Omron Sysmac Studio project asansörsonnnnnnnnnn (Sysmac Studio 1.43.0.9, StandardProject)

# Controller new_Controller_0: NJ501-1500 version 1.42
Units and slaves: Power Supply : NJ-Px3001; CPU : NJ501-1500
Task PrimaryTask (priority 4, period or condition 1000): Program0

PROGRAM Program0
VAR
    buton1 : BOOL;  (* buton1 *)
    buton2 : BOOL;  (* buton2 *)
    butonn : INT;
    buton3 : BOOL;
    kat1 : BOOL;
    sensor : INT;
    kat2 : BOOL;
    kat3 : BOOL;
    motor : INT;
    ileri : BOOL;
    geri : BOOL;
    dizi : ARRAY[0..2] OF INT;
    görev : INT;
    kapiac : BOOL;  (* kapiac *)
    kapikapa : BOOL;  (* kapikapamotor *)
    kapiacilmasüresi : TON;
    a : TIME;
    kapikapanmasüresi : TON;
    b : TIME;
    kapikapalisensör : BOOL;  (* kapikapalisensör *)
    kapiaciksensör : BOOL;  (* kapiaciksensör *)
    kapiacilmasüresi2 : TON;
    c : TIME;
    kapikapanmasüresi2 : TON;
    kapiacilmasüresi1 : TON;
    kapiacilmasüresi3 : TON;
    kapiac2 : BOOL;  (* kapiac2 *)
    kapikapa2 : BOOL;  (* kapikapa2 *)
    kapiac3 : BOOL;  (* kapiac3 *)
    kapikapa3 : BOOL;  (* kapikapa3 *)
    kapikapanmasüresi3 : TON;
END_VAR
VAR
    _p1 : BOOL;
END_VAR

(* Section Section2: ladder, written here as Structured Text *)

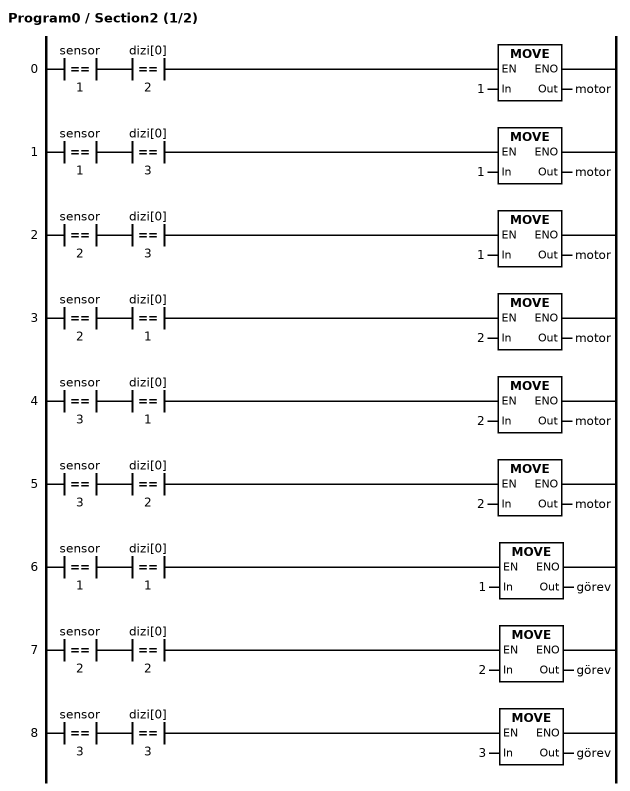
(* Rung 0 *)
IF (sensor = 1) AND (dizi[0] = 2) THEN motor := 1; END_IF;
(* Rung 1 *)
IF (sensor = 1) AND (dizi[0] = 3) THEN motor := 1; END_IF;
(* Rung 2 *)
IF (sensor = 2) AND (dizi[0] = 3) THEN motor := 1; END_IF;
(* Rung 3 *)
IF (sensor = 2) AND (dizi[0] = 1) THEN motor := 2; END_IF;
(* Rung 4 *)
IF (sensor = 3) AND (dizi[0] = 1) THEN motor := 2; END_IF;
(* Rung 5 *)
IF (sensor = 3) AND (dizi[0] = 2) THEN motor := 2; END_IF;
(* Rung 6 *)
IF (sensor = 1) AND (dizi[0] = 1) THEN görev := 1; END_IF;
(* Rung 7 *)
IF (sensor = 2) AND (dizi[0] = 2) THEN görev := 2; END_IF;
(* Rung 8 *)
IF (sensor = 3) AND (dizi[0] = 3) THEN görev := 3; END_IF;

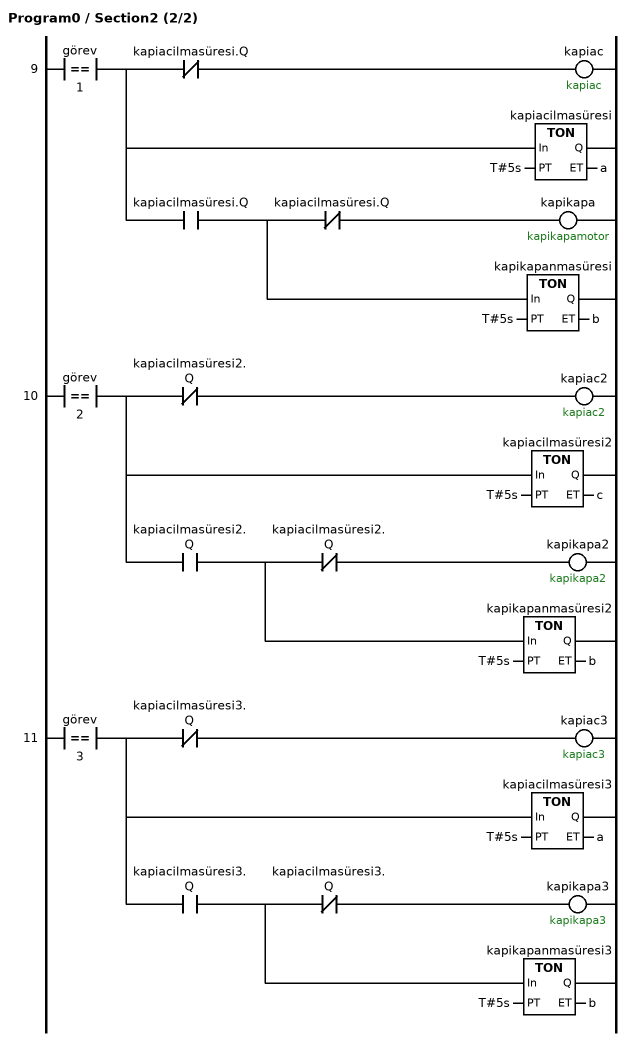
(* Rung 9 *)
kapiac := (görev = 1) AND NOT kapiacilmasüresi.Q;
kapiacilmasüresi(In := görev = 1, PT := T#5s, ET => a);
kapikapa := (görev = 1) AND kapiacilmasüresi.Q AND NOT kapiacilmasüresi.Q;
kapikapanmasüresi(In := (görev = 1) AND kapiacilmasüresi.Q, PT := T#5s, ET => b);
(* Rung 10 *)
kapiac2 := (görev = 2) AND NOT kapiacilmasüresi2.Q;
kapiacilmasüresi2(In := görev = 2, PT := T#5s, ET => c);
kapikapa2 := (görev = 2) AND kapiacilmasüresi2.Q AND NOT kapiacilmasüresi2.Q;
kapikapanmasüresi2(In := (görev = 2) AND kapiacilmasüresi2.Q, PT := T#5s, ET => b);
(* Rung 11 *)
kapiac3 := (görev = 3) AND NOT kapiacilmasüresi3.Q;
kapiacilmasüresi3(In := görev = 3, PT := T#5s, ET => a);
kapikapa3 := (görev = 3) AND kapiacilmasüresi3.Q AND NOT kapiacilmasüresi3.Q;
kapikapanmasüresi3(In := (görev = 3) AND kapiacilmasüresi3.Q, PT := T#5s, ET => b);

(* Section Section3: ladder, written here as Structured Text *)

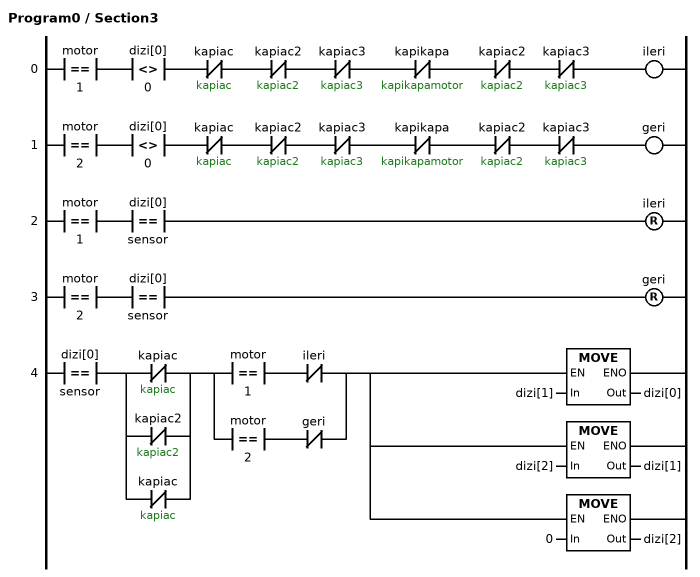
(* Rung 0 *)
ileri := (motor = 1) AND (dizi[0] <> 0) AND NOT kapiac AND NOT kapiac2 AND NOT kapiac3 AND NOT kapikapa AND NOT kapiac2 AND NOT kapiac3;
(* Rung 1 *)
geri := (motor = 2) AND (dizi[0] <> 0) AND NOT kapiac AND NOT kapiac2 AND NOT kapiac3 AND NOT kapikapa AND NOT kapiac2 AND NOT kapiac3;
(* Rung 2 *)
IF (motor = 1) AND (dizi[0] = sensor) THEN ileri := FALSE; END_IF;
(* Rung 3 *)
IF (motor = 2) AND (dizi[0] = sensor) THEN geri := FALSE; END_IF;
(* Rung 4 *)
_p1 := (dizi[0] = sensor) AND (NOT kapiac OR NOT kapiac2 OR NOT kapiac) AND (((motor = 1) AND NOT ileri) OR ((motor = 2) AND NOT geri));
IF _p1 THEN
    dizi[0] := dizi[1];
    dizi[1] := dizi[2];
    dizi[2] := 0;
END_IF;

(* Section Section1: ladder, written here as Structured Text *)

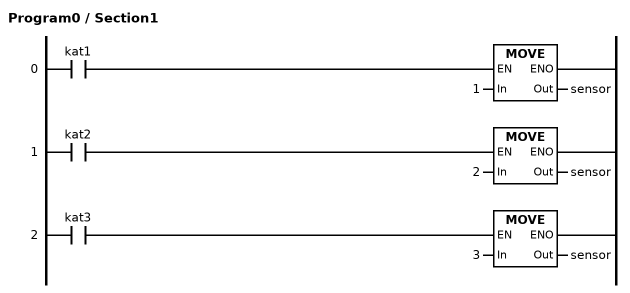
(* Rung 0 *)
IF kat1 THEN sensor := 1; END_IF;
(* Rung 1 *)
IF kat2 THEN sensor := 2; END_IF;
(* Rung 2 *)
IF kat3 THEN sensor := 3; END_IF;

(* Section Section0: ladder, written here as Structured Text *)

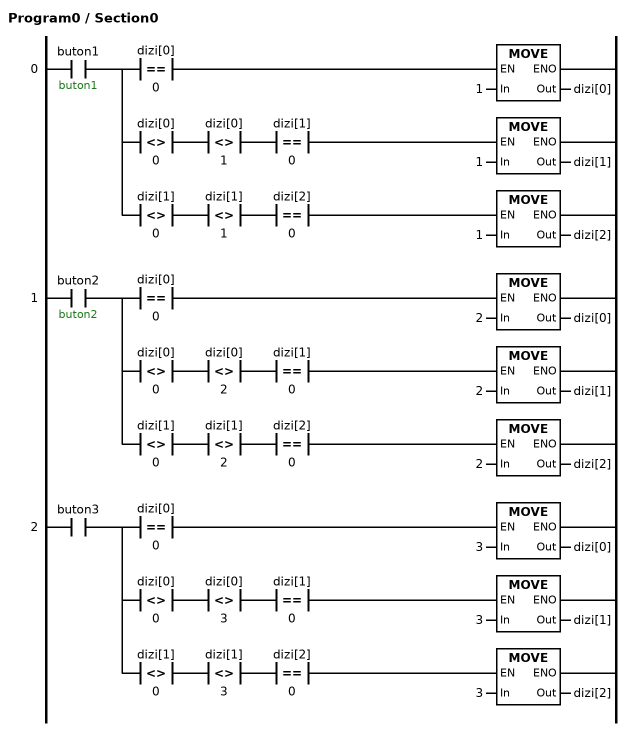
(* Rung 0 *)
IF buton1 AND (dizi[0] = 0) THEN dizi[0] := 1; END_IF;
IF buton1 AND (dizi[0] <> 0) AND (dizi[0] <> 1) AND (dizi[1] = 0) THEN dizi[1] := 1; END_IF;
IF buton1 AND (dizi[1] <> 0) AND (dizi[1] <> 1) AND (dizi[2] = 0) THEN dizi[2] := 1; END_IF;
(* Rung 1 *)
IF buton2 AND (dizi[0] = 0) THEN dizi[0] := 2; END_IF;
IF buton2 AND (dizi[0] <> 0) AND (dizi[0] <> 2) AND (dizi[1] = 0) THEN dizi[1] := 2; END_IF;
IF buton2 AND (dizi[1] <> 0) AND (dizi[1] <> 2) AND (dizi[2] = 0) THEN dizi[2] := 2; END_IF;
(* Rung 2 *)
IF buton3 AND (dizi[0] = 0) THEN dizi[0] := 3; END_IF;
IF buton3 AND (dizi[0] <> 0) AND (dizi[0] <> 3) AND (dizi[1] = 0) THEN dizi[1] := 3; END_IF;
IF buton3 AND (dizi[1] <> 0) AND (dizi[1] <> 3) AND (dizi[2] = 0) THEN dizi[2] := 3; END_IF;
END_PROGRAM